(* CoDeSys 2.3.9.28 project: Ex3 DobradorDeCantoneiras.pro *)
(* Libraries: Standard.lib 27.1.09 11:27:38, Util.lib 27.1.09 11:27:38, IecSfc.lib 24.11.08 08:07:15, SysLibTime.lib 27.1.09 11:27:38, SysTaskInfo.lib 24.11.08 08:07:15, SYSLIBCALLBACK.LIB 27.1.09 11:27:38 *)

(* PLC configuration (modules and I/O channels)
Hexswitch AT %IB0 [HexSwitch] rotary switch 0 = STOP, 1-15 = RUN
8DI/8DO [CPX-8DI_8DO_Multi_I_O_module_1] node 0, in %IB4 out %QB0 {StringParam = 4,8,1,8,1; ByteParam = 7; ByteParam = 81; ByteParam = 0; ByteParam = 0; ByteParam = 0; ByteParam = 0; ByteParam = 0; IdleStateParam = 0; IdleModeParam = 255; IdleStateParam = 0; IdleModeParam = 255; IdleStateParam = 0; IdleModeParam = 255; IdleStateParam = 0; IdleModeParam = 255}
  AT %IB4 [ByteInput] -
  AT %QB0 [ByteOutput] -
8DI/8DO [CPX-8DI_8DO_Multi_I_O_module_1] node 1, in %IB8 out %QB4 {StringParam = 4,8,1,8,1; ByteParam = 7; ByteParam = 81; ByteParam = 0; ByteParam = 0; ByteParam = 0; ByteParam = 0; ByteParam = 0; IdleStateParam = 0; IdleModeParam = 255; IdleStateParam = 0; IdleModeParam = 255; IdleStateParam = 0; IdleModeParam = 255; IdleStateParam = 0; IdleModeParam = 255}
  AT %IB8 [ByteInput] -
  AT %QB4 [ByteOutput] -
*)

(* Global variable list: Global_Variables *)
VAR_GLOBAL

	START AT  %IX2.0 : BOOL;
	STOP AT  %IX2.1 : BOOL;
	S1 AT  %IX2.2 : BOOL;
	S2 AT  %IX2.3 : BOOL;
	S3 AT  %IX2.4 : BOOL;
	S4 AT  %IX2.5 : BOOL;

	L1 AT  %QX0.0 : BOOL;
	M1 AT  %QX0.1 : BOOL;
	C1 AT  %QX0.2 : BOOL;
	C2 AT  %QX0.3 : BOOL;
	C3 AT  %QX0.4 : BOOL;

END_VAR

(* POU PLC_PRG, LD *)
PROGRAM PLC_PRG
VAR
END_VAR
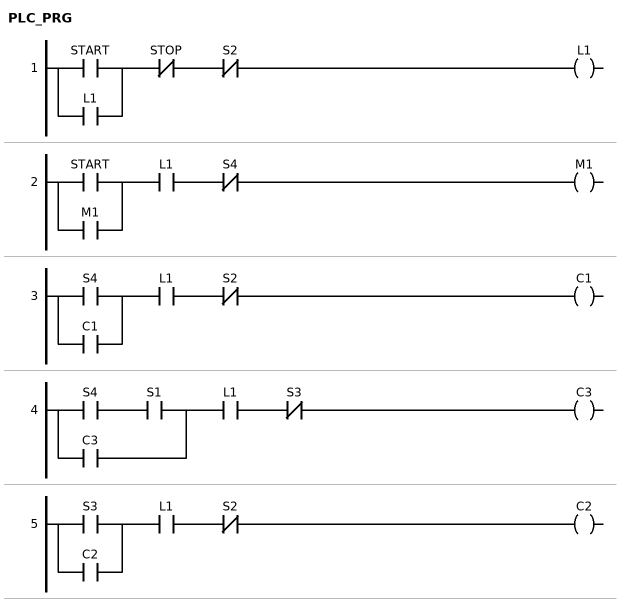
_LD_ (* Ladder Diagram *)
NETWORK 1
	{ [START] | [L1] } - [/STOP] - [/S2] --- (L1)
NETWORK 2
	{ [START] | [M1] } - [L1] - [/S4] --- (M1)
NETWORK 3
	{ [S4] | [C1] } - [L1] - [/S2] --- (C1)
NETWORK 4
	{ [S4] - [S1] | [C3] } - [L1] - [/S3] --- (C3)
NETWORK 5
	{ [S3] | [C2] } - [L1] - [/S2] --- (C2)
_END_LD_
(* the same logic as Structured Text *)
(* Network 1 *)
L1 := (START OR L1) AND NOT STOP AND NOT S2;
(* Network 2 *)
M1 := (START OR M1) AND L1 AND NOT S4;
(* Network 3 *)
C1 := (S4 OR C1) AND L1 AND NOT S2;
(* Network 4 *)
C3 := (S4 AND S1 OR C3) AND L1 AND NOT S3;
(* Network 5 *)
C2 := (S3 OR C2) AND L1 AND NOT S2;
END_PROGRAM
